(* IEC 61131-3 sources: Lasal/CPU_5344_V01/Class/positionSettingMpsControl, 1 file *)

(* ---- positionSettingMpsControl.st ---- *)
(*!
<Class
	Name               = "positionSettingMpsControl"
	Revision           = "1.0"
	RealtimeTask       = "false"
	CyclicTask         = "false"
	BackgroundTask     = "false"
	Sigmatek           = "false"
	OSInterface        = "false"
	HighPriority       = "false"
	Automatic          = "false"
	UpdateMode         = "Prescan"
	SharedCommandTable = "true"
	Objectsize         = "(284,120)">
	<Channels>
		<Server Name="setting1" Visualized="true" Initialize="false" WriteProtected="true" Retentive="false" Comment="x-pos, doesn&apos;t make sense, but also doesnt hurt&#13;&#10;"/>
		<Server Name="setting2" Visualized="true" Initialize="false" WriteProtected="false" Retentive="false" Comment="min. position (1/10e mm)"/>
		<Server Name="setting3" Visualized="true" Initialize="false" WriteProtected="false" Retentive="false" Comment="max. position (1/10e mm)"/>
		<Client Name="iMaxPos" Required="true" Internal="false"/>
		<Client Name="iMinPos" Required="true" Internal="false"/>
	</Channels>
	<Network Name="positionSettingMpsControl">
		<!-- List of Components in this network -->
		<Components>
			<Object
				Name       = "_base"
				Class      = "baseToolSettingsMpsControl"
				Position   = "(218,120)"
				Visualized = "true">
				<Channels>
					<Server Name="amountOfSettings" Value="4"/>
					<Server Name="ClassSvr"/>
					<Server Name="Name"/>
					<Server Name="plane"/>
					<Server Name="toolType" Value="1"/>
				</Channels>
			</Object>
		</Components>
		<Comments>
		</Comments>
		<!-- List of Connections in this network -->
		<Connections>
			<Connection Source="this.ClassSvr" Destination="_base.ClassSvr" Vertices="(690,210),(518,210),"/>
			<Connection Source="this.toolType" Destination="_base.toolType" Vertices="(690,270),(518,270),"/>
			<Connection Source="this.amountOfSettings" Destination="_base.amountOfSettings" Vertices="(690,450),(518,450),"/>
			<Connection Source="this.plane" Destination="_base.plane" Vertices="(690,390),(518,390),"/>
			<Connection Source="this.Name" Destination="_base.Name" Vertices="(690,330),(518,330),"/>
		</Connections>
		<!-- Headerfiles -->
		<Options>
		</Options>
	</Network>
</Class>
*)
#pragma using baseToolSettingsMpsControl

positionSettingMpsControl : CLASS
: baseToolSettingsMpsControl
  //Servers:
	setting1 	: SvrCh_DINT;
	setting2 	: SvrCh_DINT;
	setting3 	: SvrCh_DINT;
  //Clients:
	iMinPos 	: CltCh_DINT;
	iMaxPos 	: CltCh_DINT;
  //Variables:
  //Functions:

	FUNCTION VIRTUAL GLOBAL setting2::Read
		VAR_OUTPUT
			output (EAX) 	: DINT;
		END_VAR;

	FUNCTION VIRTUAL GLOBAL setting3::Read
		VAR_OUTPUT
			output (EAX) 	: DINT;
		END_VAR;
  //Tables:
	FUNCTION @STD
		VAR_OUTPUT
			ret_code	: CONFSTATES;
		END_VAR;
	FUNCTION GLOBAL TAB @CT_;
END_CLASS;

// JdK 6-2-2020: millToolSettingsMpsControl created for first test to read in settings to pc
// at this moment the class is only for storage off fixed machine data for mill tools

FUNCTION VIRTUAL GLOBAL positionSettingMpsControl::setting2::Read
	VAR_OUTPUT
		output (EAX) 	: DINT;
	END_VAR

  iMinPos:= iMinPos.Read();
  setting2:= iMinPos;
	output := setting2;

END_FUNCTION

FUNCTION VIRTUAL GLOBAL positionSettingMpsControl::setting3::Read
	VAR_OUTPUT
		output (EAX) 	: DINT;
	END_VAR

  iMaxPos:= iMaxPos.Read();
  setting3:= iMaxPos;
	output := setting3;

END_FUNCTION
